FUNCTION_BLOCK FB_BaseHMILoggerElement_View EXTENDS FB_Base IMPLEMENTS ITF_BaseHMILoggerElement_View
VAR
	itfBaseLoggerConnector					: ITF_BaseLogger_HMI_Connector_View;	//bezpośredni łącznik do logera odczyt danych
	itfBaseLoggerElementConnector			: ITF_BaseLoggerElement_HMI_Connector_View;	//lacznik do FB_BaseLoggerElement np zeby wyciągnąć identyfikator odczyt danych
	refstBaseLoggerElementDataHMI			: REFERENCE TO ST_BaseHMILoggerElement_View;
	refstMemoryEvents						: REFERENCE TO ST_BaseEvents_Memory;	//referencja do tablicy zgłoszeń
	bIsInit									: BOOL;	//flaga informująca czy wszystkie interfejsy są dobrze przypisane
	bIsValidData							: bool;	//flaga informująca czy wszystkie dane sa podpięte 
END_VAR

(*			
	RafalOS
	Rafał Osajda		19.11.2025		TC 4024.66
	Czyści danych przy zmienia ramki po poprzedniej ramce
*)
METHOD PUBLIC ClearAfterScreen : BOOL
VAR_INPUT
END_VAR
END_METHOD

METHOD PRIVATE CompleteTheDetailedInformation : BOOL
VAR_INPUT
	stRow			: ST_BaseHMIConnectorEvents_ListToDisplayRow;
END_VAR
THIS^.refstBaseLoggerElementDataHMI.stDetailInformation.uiIDEvent						:= stRow.uiIDEvent;
THIS^.refstBaseLoggerElementDataHMI.stDetailInformation.uiIDItem						:= stRow.uiIDItem;
THIS^.refstBaseLoggerElementDataHMI.stDetailInformation.sCode							:= stRow.sCode;
THIS^.refstBaseLoggerElementDataHMI.stDetailInformation.bActive							:= stRow.bActive;
THIS^.refstBaseLoggerElementDataHMI.stDetailInformation.bIgnoreRepetitions				:= stRow.bIgnoreRepetitions;
THIS^.refstBaseLoggerElementDataHMI.stDetailInformation.uiRepetitionCounter				:= stRow.uiRepetitionCounter;
THIS^.refstBaseLoggerElementDataHMI.stDetailInformation.sStart							:= stRow.sStart;
THIS^.refstBaseLoggerElementDataHMI.stDetailInformation.sFinish							:= stRow.sFinish;
THIS^.refstBaseLoggerElementDataHMI.stDetailInformation.sConfirmed						:= stRow.sConfirmed;
THIS^.refstBaseLoggerElementDataHMI.stDetailInformation.bConfirm						:= stRow.bConfirm;
THIS^.refstBaseLoggerElementDataHMI.stDetailInformation.bConfirmed						:= stRow.bConfirmed;
THIS^.refstBaseLoggerElementDataHMI.stDetailInformation.sEventCategory					:= stRow.sEventCategory;
THIS^.refstBaseLoggerElementDataHMI.stDetailInformation.wsDescription					:= stRow.wsDescription;
THIS^.refstBaseLoggerElementDataHMI.stDetailInformation.wsDescriptionFull				:= stRow.wsDescriptionFull;
END_METHOD

METHOD PRIVATE CopyDataToDisplay : BOOL
VAR_INPUT
	refarrToDisplay				: REFERENCE TO ARRAY [1..GVL_BaseConstans.MAX_EVENTS_TO_SHOW] OF ST_BaseHMIConnectorEvents_ListToDisplayRow;
	iNumberOfRow				: INT;
	stRowFromMemory				: ST_BaseEvents_RowInMemory;
	stItemInformation			: ST_BaseLogger_ItemDataToDisplay;
END_VAR
VAR
	wstmpDescriptionFull		: WSTRING;
	wstmpDescription			: WSTRING;
	iDltmp						: INT;
END_VAR
refarrToDisplay [iNumberOfRow].uiIDEvent			:= stRowFromMemory.uiIDEvent;
refarrToDisplay [iNumberOfRow].uiIDItem				:= stRowFromMemory.uiIDItem;
refarrToDisplay [iNumberOfRow].bActive				:= stRowFromMemory.bActive;
refarrToDisplay [iNumberOfRow].sCode				:= stItemInformation.sCode; 
refarrToDisplay [iNumberOfRow].bIgnoreRepetitions	:= stRowFromMemory.bIgnoreRepetitions;
refarrToDisplay [iNumberOfRow].bConfirm				:= stRowFromMemory.bConfirm;
refarrToDisplay [iNumberOfRow].bConfirmed			:= stRowFromMemory.bConfirmed;

refarrToDisplay [iNumberOfRow].sStart				:= THIS^.refstCommonData.itfTime.BaseDTToString (inDT := stRowFromMemory.dtStart);
IF (TO_STRING (stRowFromMemory.dtConfirmed) <> 'DT#1970-01-01-00:00:00') THEN
	refarrToDisplay [iNumberOfRow].sConfirmed		:= THIS^.refstCommonData.itfTime.BaseDTToString (inDT := stRowFromMemory.dtConfirmed);
ELSE
	refarrToDisplay [iNumberOfRow].sConfirmed		:= '';
END_IF
IF (TO_STRING (TO_STRING (stRowFromMemory.dtFinish)) <> 'DT#1970-01-01-00:00:00') THEN
	refarrToDisplay [iNumberOfRow].sFinish			:= THIS^.refstCommonData.itfTime.BaseDTToString (inDT := stRowFromMemory.dtFinish);
ELSE
	refarrToDisplay [iNumberOfRow].sFinish			:= '';
END_IF

refarrToDisplay [iNumberOfRow].sEventCategory		:= stItemInformation.sEventCategory; 
refarrToDisplay [iNumberOfRow].uiRepetitionCounter	:= stItemInformation.uiRepetitionCounter;
wstmpDescriptionFull		:= THIS^.GetTextFromLabelForActiveLocation (stLabel	:= stItemInformation.stDescription);
iDltmp												:= WLEN (wstmpDescriptionFull);
IF (iDltmp > 100) THEN
	wstmpDescription								:= WDELETE (wstmpDescriptionFull, iDltmp - 100, iDltmp);
END_IF
refarrToDisplay [iNumberOfRow].wsDescription		:= wstmpDescription;
refarrToDisplay [iNumberOfRow].wsDescriptionFull	:= wstmpDescriptionFull;
refarrToDisplay [iNumberOfRow].wsNameOfitem			:= THIS^.GetTextFromLabelForActiveLocation (stLabel := stItemInformation.stItemName);
END_METHOD

METHOD PUBLIC CreateLinkToEventsMemory : BOOL
VAR_INPUT
END_VAR
THIS^.refstMemoryEvents	REF= THIS^.itfBaseLoggerConnector.GetReferenceToStmemory ();


IF (__ISVALIDREF (THIS^.refstMemoryEvents)) THEN
	CreateLinkToEventsMemory		:= TRUE;
ELSE
	CreateLinkToEventsMemory		:= FALSE;
END_IF
END_METHOD

(*			
	EVERDE sp. z o.o.
	Rafał Osajda		09.09.2025		TC 4024.66
	Generuje tablicę zdarzeń dla podanego ID dla 0 dla wszystkich elementów
*)
METHOD PUBLIC GetEventTableForIDItem : BOOL
VAR_INPUT
	uiIdItem				: UINT;
END_VAR
VAR_INST
	bFilterIsActivePrevius	: BOOL;	
END_VAR
VAR
	iI						: INT;
	bFilterIsActive			: BOOL;
	bUsunZListy				: BOOL;
	btmpUsunZListy			: BOOL;
	refstMemory				: REFERENCE TO ST_BaseEvents_Memory;
	refstListToDisplay		: REFERENCE TO ST_BaseHMIConnectorEvents_ListToDisplay;
	refstFilter				: REFERENCE TO ST_BaseHMIConnectorEvents_Filter;
	refstActionButtons		: REFERENCE TO ST_BaseHMIConnectorEvents_ActionButtuns;
	stRowFromMemory			: ST_BaseEvents_RowInMemory;
	stItemInformation		: ST_BaseLogger_ItemDataToDisplay;
(*	Ilosci zdarzen wyswietlanych na liscie	*)
	stNumberEventToDisplay	: ST_BaseEvents_ActiveEvents;
//
	iIAck: INT;
	iIClose: INT;
END_VAR
(*
	sprawdzenie czy jest coś nowego - tak generuj
	jak już jest wygenerowana jakaś lista i zmienił się filtr - tak to generuj

*)
IF (THIS^.refstMemoryEvents.iNumberOfRow > 0) THEN

	refstMemory				REF= THIS^.refstMemoryEvents;
	refstListToDisplay		REF= THIS^.refstBaseLoggerElementDataHMI.stListOfEventsToDisplay;
	refstFilter				REF= THIS^.refstBaseLoggerElementDataHMI.stFilter;
	refstActionButtons		REF= THIS^.refstBaseLoggerElementDataHMI.stButtons;
	bFilterIsActive			:= GetIsActiveFilter (refstFilter := refstFilter);		//sprawdzenie czy jest aktywny filtr
	
	IF (THIS^.itfBaseLoggerConnector.GetChangeInMemory () OR bFilterIsActive 
		OR bFilterIsActivePrevius OR THIS^.refstBaseLoggerElementDataHMI.bRefreshList) THEN
		THIS^.refstBaseLoggerElementDataHMI.bRefreshList	:= FALSE;
		bFilterIsActivePrevius								:= bFilterIsActive;

		THIS^.itfBaseLoggerConnector.ResetChangeInMemory ();
		(*	Wyczyszczenie tablicy wyświetlania		*)
		Tc2_System.MEMSET (
			destAddr		:= ADR (refstListToDisplay.arrToDisplay),
			fillByte		:= 0,
			n				:= SIZEOF (refstListToDisplay.arrToDisplay)
		);
		refstListToDisplay.iNumberOfRow		:= 0;
		FOR iI := 1 TO refstMemory.iNumberOfRow DO
			IF (uiIdItem = refstMemory.arrRow [iI].uiIDItem OR uiIdItem = 0) THEN
				stRowFromMemory			:= refstMemory.arrRow [iI];
				stItemInformation		:= THIS^.itfBaseLoggerConnector.GetInformationFromItem (uiIDItem := uiIdItem, uiIDEvent := stRowFromMemory.uiIDEvent);
				bUsunZListy		:= THIS^.RemoveRowFormList (
										refstFilter 		:= refstFilter, 
										uiIDEvent 			:= stRowFromMemory.uiIDEvent, 
										uiIDItem 			:=  stRowFromMemory.uiIDItem,
										bActive				:= stRowFromMemory.bActive,
										stItemInformation	:= stItemInformation
									);
				IF (NOT bUsunZListy) THEN
					refstListToDisplay.iNumberOfRow		:= refstListToDisplay.iNumberOfRow + 1;
					THIS^.CopyDataToDisplay (
						refarrToDisplay					:= refstListToDisplay.arrToDisplay,
						iNumberOfRow					:= refstListToDisplay.iNumberOfRow,
						stRowFromMemory					:= stRowFromMemory,
						stItemInformation				:= stItemInformation
					);
	(*	Informacja o ilosciach zgloszen na wyswietlanej liście 		*)
					stNumberEventToDisplay.iTotalNumer	:= stNumberEventToDisplay.iTotalNumer + 1;
					IF (refstListToDisplay.arrToDisplay [refstListToDisplay.iNumberOfRow].bActive) THEN
						stNumberEventToDisplay.iNumberOfActive	:= stNumberEventToDisplay.iNumberOfActive + 1;
						stNumberEventToDisplay.arrNumberOfActive [stItemInformation.eEventCategory] := stNumberEventToDisplay.arrNumberOfActive [stItemInformation.eEventCategory] + 1;
						stNumberEventToDisplay.arrActive [stItemInformation.eEventCategory]	:= TRUE;
					END_IF
					IF (refstListToDisplay.arrToDisplay [refstListToDisplay.iNumberOfRow].bConfirm AND 
						NOT refstListToDisplay.arrToDisplay [refstListToDisplay.iNumberOfRow].bConfirmed) THEN
						stNumberEventToDisplay.iNumberOfActiveWithConfirmation	:= stNumberEventToDisplay.iNumberOfActiveWithConfirmation + 1;
					END_IF
					stNumberEventToDisplay.arrTotalNumer [stItemInformation.eEventCategory] := stNumberEventToDisplay.arrTotalNumer [stItemInformation.eEventCategory] + 1;
				END_IF	//usuwanie z listy
			END_IF
	(*	Liczba zgłoszeń większa od tych co wyświetlamy	starsze można zobaczyć na kompie po podłaczeniu 	*)
			IF (refstListToDisplay.iNumberOfRow = TO_INT (GVL_BaseConstans.MAX_EVENTS_TO_SHOW)) THEN
				EXIT;
			END_IF
		END_FOR	//koniec przechodzenia przez wiersze pamięci
	(*	Informacja o ilosciach zgloszen		*)
		IF (uiIdItem > 0) THEN
			THIS^.PrepareQuantitiesForDisplay (
				stCounted		:= stNumberEventToDisplay,
				stFromLogger	:= THIS^.itfBaseLoggerConnector.GetEventCountsForItem (uiIDItem := uiIDItem)
			);
		ELSE
			THIS^.PrepareQuantitiesForDisplay (
				stCounted		:= stNumberEventToDisplay,
				stFromLogger	:= THIS^.itfBaseLoggerConnector.GetEventCounts ()
			);
		END_IF
		refstActionButtons.bAcknowledgeAllActive	:= stNumberEventToDisplay.iNumberOfActiveWithConfirmation > 0;
		refstActionButtons.bCloseAllActive			:= stNumberEventToDisplay.iNumberOfActive > 0;
	END_IF
	IF (THIS^.refstBaseLoggerElementDataHMI.bSelected) THEN
		refstActionButtons.bAcknowledgeSelectedActive	:= refstListToDisplay.arrToDisplay [THIS^.refstBaseLoggerElementDataHMI.iSelectedRow].bConfirm AND 
			NOT refstListToDisplay.arrToDisplay [THIS^.refstBaseLoggerElementDataHMI.iSelectedRow].bConfirmed;
		refstActionButtons.bCloseSelectedActive			:= refstListToDisplay.arrToDisplay [THIS^.refstBaseLoggerElementDataHMI.iSelectedRow].bConfirm AND 
			refstListToDisplay.arrToDisplay [THIS^.refstBaseLoggerElementDataHMI.iSelectedRow].bConfirmed;
	ELSE
		refstActionButtons.bAcknowledgeSelectedActive	:= FALSE;
		refstActionButtons.bCloseSelectedActive			:= FALSE;
	END_IF
	
	(*	Wybor zgloszenia z listy	*)

	IF ((THIS^.refstBaseLoggerElementDataHMI.iSelectedRow <> THIS^.refstBaseLoggerElementDataHMI.iSelectedRowPrevius AND
		THIS^.refstBaseLoggerElementDataHMI.bSelected) OR THIS^.refstBaseLoggerElementDataHMI.bRefreshInfo ) THEN
		THIS^.CompleteTheDetailedInformation (stRow := refstListToDisplay.arrToDisplay [THIS^.refstBaseLoggerElementDataHMI.iSelectedRow]);
	ELSIF (NOT THIS^.refstBaseLoggerElementDataHMI.bSelected) THEN
		THIS^.refstBaseLoggerElementDataHMI.iSelectedRow		:= -1;
		THIS^.refstBaseLoggerElementDataHMI.iSelectedRowPrevius	:= -1;
	END_IF 
	
	(*	Obsługa przycisków zamykania i potwierrdzania zgłoszeń	*)

	IF (THIS^.refstBaseLoggerElementDataHMI.stButtons.bAcknowledgeSelected) THEN //potwierdz zgłoszenie
		IF (refstListToDisplay.arrToDisplay [THIS^.refstBaseLoggerElementDataHMI.iSelectedRow].bConfirm AND 
			NOT refstListToDisplay.arrToDisplay [THIS^.refstBaseLoggerElementDataHMI.iSelectedRow].bConfirmed) THEN
			THIS^.itfBaseLoggerElementConnector.EventAcknowledgeByID (uiIDEvent := THIS^.refstBaseLoggerElementDataHMI.stDetailInformation.uiIDEvent);
		END_IF
	END_IF

	IF (THIS^.refstBaseLoggerElementDataHMI.stButtons.bCloseSelected) THEN	//zamknij zgłoszenie
		IF (refstListToDisplay.arrToDisplay [THIS^.refstBaseLoggerElementDataHMI.iSelectedRow].bActive OR 
			refstListToDisplay.arrToDisplay [THIS^.refstBaseLoggerElementDataHMI.iSelectedRow].sFinish <> '') THEN
			THIS^.itfBaseLoggerElementConnector.EventSetInactiveByID (uiIDEvent := THIS^.refstBaseLoggerElementDataHMI.stDetailInformation.uiIDEvent);
		END_IF
	END_IF

	IF (THIS^.refstBaseLoggerElementDataHMI.stButtons.bAcknowledgeAll) THEN //potwierdz wszystkie niepotwierdzone zgłoszenie
		FOR iIAck := 1 TO TO_INT (refstListToDisplay.iNumberOfRow) DO
			IF (refstListToDisplay.arrToDisplay [iIAck].bConfirm AND 
				NOT refstListToDisplay.arrToDisplay [iIAck].bConfirmed) THEN
				THIS^.itfBaseLoggerElementConnector.EventAcknowledgeByID (uiIDEvent := refstListToDisplay.arrToDisplay [iIAck].uiIDEvent);
			END_IF
		END_FOR
	END_IF
	IF (THIS^.refstBaseLoggerElementDataHMI.stButtons.bCloseAll) THEN	//zamknij wszystkie nie zamnknięte zgłoszenie
		FOR iIClose := 1 TO TO_INT (refstListToDisplay.iNumberOfRow) DO
			IF (refstListToDisplay.arrToDisplay [iIClose].bActive OR refstListToDisplay.arrToDisplay [iIClose].sFinish <> '') THEN
				THIS^.itfBaseLoggerElementConnector.EventSetInactiveByID (uiIDEvent := refstListToDisplay.arrToDisplay [iIClose].uiIDEvent);
			END_IF
		END_FOR
	END_IF
	
	
	THIS^.refstBaseLoggerElementDataHMI.bRefreshList		:= 	refstActionButtons.bAcknowledgeSelected OR
																refstActionButtons.bCloseSelected OR
																refstActionButtons.bAcknowledgeAll OR
																refstActionButtons.bCloseAll;
	THIS^.refstBaseLoggerElementDataHMI.bRefreshInfo		:= 	refstActionButtons.bAcknowledgeSelected	OR
																refstActionButtons.bCloseSelected OR
	                                                          	refstActionButtons.bAcknowledgeAll OR
                                                               	refstActionButtons.bCloseAll;
	refstActionButtons.bAcknowledgeSelected					:= FALSE;
	refstActionButtons.bCloseSelected						:= FALSE;
	refstActionButtons.bAcknowledgeAll						:= FALSE;
	refstActionButtons.bCloseAll							:= FALSE;

END_IF
END_METHOD

METHOD PRIVATE GetIsActiveFilter : BOOL
VAR_INPUT
	refstFilter				: REFERENCE TO ST_BaseHMIConnectorEvents_Filter;
END_VAR
VAR
	bResult: BOOL;
	iI: INT;
END_VAR
bResult				:= refstFilter.bActive OR 
						refstFilter.bNotActive OR
						refstFilter.bIDEvent OR
						refstFilter.bIDItem;
FOR iI := 1 TO GVL_BaseConstans.NUMBER_OF_EVENT_CATEGORIES DO
	bResult			:= bResult OR refstFilter.arrSelectedEventCategory [iI];
END_FOR

GetIsActiveFilter	:= bResult;
END_METHOD

METHOD PROTECTED GetTextFromLabel : WSTRING
VAR_INPUT
	stLabel				: ST_BaseLabel;
	eLocation			: E_BaseLocation;
END_VAR
GetTextFromLabel := stLabel.arrText [eLocation];
END_METHOD

METHOD PROTECTED GetTextFromLabelForActiveLocation : WSTRING
VAR_INPUT
	stLabel				: ST_BaseLabel;
END_VAR

VAR
	dfsfsdaf: WSTRING;
END_VAR
GetTextFromLabelForActiveLocation := stLabel.arrText [THIS^.refstCommonData.itfLocaciotn.GetLocation ()];
END_METHOD

(*			
	EVERDE sp. z o.o.
	Rafał Osajda		09.09.2025		TC 4024.66
	Zwraca tablicę swoich zdarzeń
*)
METHOD PUBLIC GetYourEventTable : BOOL
VAR_INPUT
END_VAR
THIS^.GetEventTableForIDItem (uiIdItem := THIS^.itfBaseLoggerElementConnector.GetID ());		//przygotowanie tablicy dla siebie
END_METHOD

(*			
	RAFALOS
	Rafał Osajda		23.09.2025		TC 4024.66
	Zwraca informację czy dane są podpięte do systemu
*)
METHOD PUBLIC IsInit : BOOL
VAR_INPUT
END_VAR
IsInit			:= THIS^.bIsInit;
END_METHOD

METHOD PUBLIC IsLinkedReferences : BOOL
VAR_INPUT
END_VAR
IF (__ISVALIDREF (THIS^.refstBaseLoggerElementDataHMI)) THEN
	IsLinkedReferences			:= TRUE;
END_IF
END_METHOD

(*			
	RAFALOS
	Rafał Osajda		23.09.2025		TC 4024.66
	Zwraca flagę przypisywaną w FB_Init tworzonego elementu
*)
METHOD IsValidData : BOOL
VAR_INPUT
END_VAR
IsValidData				:= THIS^.bIsValidData;
END_METHOD

(*			
	RafalOS
	Rafał Osajda		14.11.2025		TC 4024.66
	Metoda przygotowywania danych dla HMI 
	W niej odbywa się odpytywanie właściego elementu przez łącznik
*)
METHOD PUBLIC PrepareDataForHMI : BOOL
VAR_INPUT
END_VAR
END_METHOD

(*			
	RafalOS
	Rafał Osajda		19.11.2025		TC 4024.66
	Przygotowanie ramki pood tamke do wyświetlenia - tylko przygotowanie a nie przygotowanie danych do wyświetlenia
*)
METHOD PUBLIC PrepareForScreen : BOOL
VAR_INPUT
END_VAR
END_METHOD

METHOD PRIVATE PrepareQuantitiesForDisplay : BOOL
VAR_INPUT
	stCounted			: ST_BaseEvents_ActiveEvents;
	stFromLogger		: ST_BaseEvents_ActiveEvents;
END_VAR

VAR
	iI: INT;
	stmp1: STRING;
END_VAR
stmp1	:= CONCAT (stmp1,TO_STRING (stCounted.iNumberOfActiveWithConfirmation));
stmp1	:= CONCAT (stmp1, '/');
stmp1	:= CONCAT (stmp1, TO_STRING (stFromLogger.iNumberOfActiveWithConfirmation));

THIS^.refstBaseLoggerElementDataHMI.stButtons.sAcknowledgeAll		:= stmp1;
THIS^.refstBaseLoggerElementDataHMI.stButtons.sAcknowledgeSelected	:= '1/1';

stmp1	:= CONCAT ('',TO_STRING (stCounted.iNumberOfActive));
stmp1	:= CONCAT (stmp1, '/');
stmp1	:= CONCAT (stmp1, TO_STRING (stFromLogger.iNumberOfActive));
THIS^.refstBaseLoggerElementDataHMI.stButtons.sCloseAll				:= stmp1;
THIS^.refstBaseLoggerElementDataHMI.stButtons.sCloseSelected		:= '1/1';

FOR iI := 1	TO GVL_BaseConstans.NUMBER_OF_EVENT_CATEGORIES DO
	THIS^.refstBaseLoggerElementDataHMI.stFilter.arrTextOnEventCategory [iI]	:= 
		CONCAT (TO_STRING (stCounted.arrTotalNumer [iI]), CONCAT ('/',TO_STRING (stFromLogger.arrTotalNumer [iI])));
END_FOR
END_METHOD

METHOD PRIVATE RemoveRowFormList : BOOL
VAR_INPUT
	refstFilter				: REFERENCE TO ST_BaseHMIConnectorEvents_Filter;
	uiIDEvent				: UINT;
	uiIDItem				: UINT;
	bActive					: BOOL;
	stItemInformation		: ST_BaseLogger_ItemDataToDisplay;
END_VAR
VAR
	bRemove					: BOOL;
	iK						: INT;
	bRemoveHelp				: BOOL;
END_VAR
bRemove		:= FALSE;
bRemove		:= bRemove OR (refstFilter.bActive AND NOT bActive);
bRemove		:= bRemove OR (refstFilter.bNotActive AND bActive);
bRemove		:= bRemove OR (refstFilter.bIDItem	AND uiIDItem <> refstFilter.uiIDItem);
bRemove		:= bRemove OR (refstFilter.bIDEvent AND 
uiIDEvent <> refstFilter.uiIDEvent);
FOR iK := 1 TO GVL_BaseConstans.NUMBER_OF_EVENT_CATEGORIES DO
	CASE iK OF 
		E_BaseEvents_Category.Error		: bRemoveHelp	:=  stItemInformation.eEventCategory = E_BaseEvents_Category.Error;
		E_BaseEvents_Category.Alarm		: bRemoveHelp	:=  stItemInformation.eEventCategory = E_BaseEvents_Category.Alarm;
		E_BaseEvents_Category.Safety	: bRemoveHelp	:=  stItemInformation.eEventCategory = E_BaseEvents_Category.Safety;
		E_BaseEvents_Category.Message	: bRemoveHelp	:=  stItemInformation.eEventCategory = E_BaseEvents_Category.Message;
	END_CASE
	bRemove		:= bRemove OR (refstFilter.arrSelectedEventCategory [iK] AND bRemoveHelp);
END_FOR
//przeddział czasowy

RemoveRowFormList	:= bRemove;
END_METHOD

METHOD PROTECTED SelectLocation : WSTRING
VAR_INPUT
	stTexts			: ST_BaseLabel;
	eLocation		: E_BaseLocation;
END_VAR
SelectLocation := stTexts.arrText [eLocation];
END_METHOD

END_FUNCTION_BLOCK

(* stored: Version 1.1.0.1
   POU FB_BaseHMILoggerElement_View: Id {024becb4-36e5-0a14-1436-0e8a32c5de12}, SpecialFunc None
   Folder ITF_BaseLoggerElement_HMI: Id {490d29d6-def9-07f2-16cf-bb21a6440bb9}
   Folder WiazanieZmiennych: Id {4d450796-b575-0397-39db-94123d6241c4}
   Method ClearAfterScreen: Id {17479a5b-b734-05e1-2331-97f746fc52fa}
   Method CompleteTheDetailedInformation: Id {0b06bff0-7255-0a63-19f0-5ecb92dff9d6}
   Method CopyDataToDisplay: Id {75592a02-6e87-039e-0670-1b22f05f769c}
   Method CreateLinkToEventsMemory: Id {95a4fe1d-262b-028d-22e6-1fe12c2c7cc8}
   Method GetEventTableForIDItem: Id {d7402387-758c-09da-06b8-6d4ae8c9312e}
   Method GetIsActiveFilter: Id {79a84ee2-6eaf-0e54-0e23-81a9e7b0b6f8}
   Method GetTextFromLabel: Id {a9b62345-93c3-08b6-28c4-c9ac0ac3d039}
   Method GetTextFromLabelForActiveLocation: Id {a64a1e4e-c601-06e6-195a-7e58002b1474}
   Method GetYourEventTable: Id {368f0f11-8005-0717-354f-559c5b808c9c}
   Method IsInit: Id {ff032025-bb47-0541-2e34-4756feab4ddd}
   Method IsLinkedReferences: Id {0bb5653a-e044-0c0e-035c-5823debef6f0}
   Method IsValidData: Id {f2f46b20-d299-05ed-341f-5d54b19130b7}
   Method PrepareDataForHMI: Id {331b6ebd-d5ed-0e5c-2e82-348a492deb20}
   Method PrepareForScreen: Id {a782b09d-bac8-034d-0cad-2d6d75d40276}
   Method PrepareQuantitiesForDisplay: Id {4a51ff7a-bc42-01f0-2da8-11249a1d4598}
   Method RemoveRowFormList: Id {c7b91807-0b82-0e52-2df4-6abf6578c8bd}
   Method SelectLocation: Id {6bed02d4-9bbe-0541-2dba-6a636b08d172} *)
